FUNCTION_BLOCK ABSTRACT FBA_LinearDrive IMPLEMENTS I_LinearDrive
VAR_INPUT
	bEnable : BOOL;
	sensorDefaultState : BOOL;
END_VAR
VAR_OUTPUT	
	ready : BOOL;
END_VAR
VAR
	direction : MC_Direction;
	
	step : Homing;
	homingComplete : BOOL;
	
	home AT %I* : BOOL;
END_VAR

PROPERTY ABSTRACT Active : BOOL
GET
END_GET
END_PROPERTY

{attribute 'monitoring':='call'}
PROPERTY AtHome : BOOL
GET
AtHome := home <> sensorDefaultState;
END_GET
END_PROPERTY

PROPERTY ABSTRACT Error : BOOL
GET
END_GET
END_PROPERTY

{attribute 'monitoring':='call'}
PROPERTY HomeSet : BOOL
GET
HomeSet := homingComplete;
END_GET
END_PROPERTY

METHOD ABSTRACT homingSequence : BOOL
VAR_INPUT
END_VAR
END_METHOD

METHOD ABSTRACT reset : BOOL
VAR_INPUT
END_VAR
END_METHOD

METHOD ABSTRACT stop : BOOL
VAR_INPUT
END_VAR
END_METHOD

METHOD ABSTRACT toHome : BOOL
VAR_INPUT
END_VAR
END_METHOD

END_FUNCTION_BLOCK

(* stored: Version 1.1.0.1, ProductVersion 3.1.4024.11
   POU FBA_LinearDrive: Id {623d372e-720b-492b-b1ee-c6bb52096993}, SpecialFunc None
   Folder Abstract: Id {0d969d73-dc4d-48df-acd3-9dea97aa2393}
   Folder Properties: Id {3fbcce79-23f6-4884-b543-809de5ac65d5}
   Property Active: Id {c266dd51-3e5c-4ae4-9da1-835becf6473e}
   Get Get: Id {f9d0e146-aa9f-494e-9080-866e153da66f}
   Property AtHome: Id {5f7886d2-117c-40b9-8863-b31a64a2acbe}
   Get Get: Id {bb2756ff-cb99-40de-b6c2-4ac21d390403}
   Property Error: Id {1ec6eeb7-3964-4d67-840d-0c2d03bd4972}
   Get Get: Id {b6a4e69a-b3df-4b8d-a38c-f43554a7a44d}
   Property HomeSet: Id {052febb7-84f9-4e63-9cb7-13d3e938f72e}
   Get Get: Id {86e762c4-866b-4c99-896b-5a66f762ca56}
   Method homingSequence: Id {1e78c0c5-581b-4a02-86a3-526e6f4a3708}
   Method reset: Id {fce15429-5d27-4401-b60d-28867cdef3f3}
   Method stop: Id {1c5d7548-bb12-4554-8d20-2a3d2e9f9379}
   Method toHome: Id {ce770cf5-1e30-4bd8-98fb-f0523aabf66d} *)
